FUNCTION_BLOCK FB_PrintPositionWeu EXTENDS FB_BasePrint IMPLEMENTS I_Simulation
VAR_INPUT
  IlEncoderPulse      AT%I* : UDINT;                // Encoder counter intput
  IbEncoderWcState    AT%I* : BOOL;                 // Encoder EL5101 WcState
END_VAR
VAR_OUTPUT
  bStarted                  : BOOL;                 // position started moving
  bMoving                   : BOOL;                 // position is moving
END_VAR
// ----------------------------------
// configuration
VAR
  // configuration (init)
  _fPrintResolution         : LREAL := 600;         // print(head) resolution in [dpi]
  _fSubPxResolution         : LREAL := 32;          // SubPixel resolution [SubPx], resolution factor (fI_PrintResolution*fI_SubPxResolution=>Output resolution)
  _fTaskCycleTime           : LREAL := 0.002;        // Task cycle time in [s]
END_VAR
VAR PERSISTENT
  // config values changable during runtime (recipe, visu, property)
  _fEncoderResolution       : LREAL := 1;     // Encoder resolution
END_VAR
VAR CONSTANT
  fC_MinSpeed               : LREAL := 0.05;
END_VAR
// ---------------------------------
// internal variables
VAR
  // fb inst
  //fbPositionMaster          : FB_PositionMaster;
  Fb_Ph_Master                : FB_POSITION_MASTER;
  Fb_Ref_Master               : FB_POSITION_MASTER;
  Fb_Aux_Master               : FB_POSITION_MASTER;
  
  // internal vars
  fEncoderReso              : LREAL;                // used encoder resolution
  rTrigMoving               : R_TRIG;
  // simulation
  _bSim                     : BOOL;
  rfTrig_Sim                : RF_TRIG;
    
  // test functions

END_VAR

rfTrig_Sim(CLK:=_bSim);
IF rfTrig_Sim.RT THEN SimEnter(); END_IF
IF rfTrig_Sim.FT THEN SimExit(); END_IF
IF _bSim THEN SimUpdate(); END_IF

// set internal used resolution
fEncoderReso := _fEncoderResolution;  

// calc position / speed
(*Reference Master (Used in Endless Mode with drift compensation)*)
(*---input---*)
Fb_Ref_Master.pI_ConversionErr       := ADR(PRG_SYSTEMBASE.lI_ConversionErr);
Fb_Ref_Master.bI_Reset               := bI_HardwareSync[ePr_PG_GROUP_1];  (*AutoReset*)
Fb_Ref_Master.lI_Reference           := lL_EncPulse[iL_I];
Fb_Ref_Master.fI_ResolutionInput     := fEncoderReso;
Fb_Ref_Master.fI_ResolutionOutPh     := iL_ResolutionPhPx[iL_I];
Fb_Ref_Master.fI_ResolutionOutSubPx  := iL_ResolutionSubPx[iL_I];

(*---call---*)
Fb_Ref_Master();


(*Aux Master (Used for machine speed info)*)
(*---input---*)
Fb_Aux_Master.pI_ConversionErr       := ADR(PRG_SYSTEMBASE.lI_ConversionErr);
Fb_Aux_Master.bI_Reset               := bI_HardwareSync[ePr_PG_GROUP_1];  (*AutoReset*)
Fb_Aux_Master.lI_Reference           := lIKp_EncPulse;
Fb_Aux_Master.fI_ResolutionInput     := fEncoderReso;
Fb_Aux_Master.fI_ResolutionOutPh     := iL_ResolutionPhPx[iL_I];
Fb_Aux_Master.fI_ResolutionOutSubPx  := iL_ResolutionSubPx[iL_I];

(*---call---*)
Fb_Aux_Master();


(*Printhead Master / Scaling from encoder pulses to subpixels*)
(*---input---*)
Fb_Ph_Master.pI_ConversionErr       := ADR(PRG_SYSTEMBASE.lI_ConversionErr);
Fb_Ph_Master.bI_Reset               := bI_HardwareSync[ePr_PG_GROUP_1];  (*AutoReset*)
Fb_Ph_Master.lI_Reference           := lL_EncPulse[iL_I];
Fb_Ph_Master.fI_ResolutionInput     := fL_ResolutionEncoder[iL_I] * fB_DriftControl[iL_I].fO_SpeedCorrectionFactor;
Fb_Ph_Master.fI_ResolutionOutPh     := iL_ResolutionPhPx[iL_I];
Fb_Ph_Master.fI_ResolutionOutSubPx  := iL_ResolutionSubPx[iL_I];

(*---call---*)
Fb_Ph_Master();


// postion status
bMoving := Fb_Ph_Master.fO_Master_Speed >= fC_MinSpeed; 
rTrigMoving(CLK:=bMoving);   // create started trigger output
bStarted := rTrigMoving.Q; //OR Fb_Ph_Master.bSyncReq;

PROPERTY bSimEnable : BOOL
GET
bSimEnable := _bSim;
END_GET
SET
_bSim := bSimEnable;
END_SET
END_PROPERTY

(*
  Get current "default" position.
  [SubPx] as return value and [um] as output
  :return: position in SubPx resolution
*)
METHOD getPosition : DINT
VAR_OUTPUT
  nPosition_px       : DINT;                 // Master position in [px]
  fPosition_um       : LREAL;                // Master position in [um]
END_VAR
getPosition := fbPositionMaster.lMasterPosition;
nPosition_px := fbPositionMaster.lMasterPosition / LREAL_TO_DINT(_fSubPxResolution);
fPosition_um := fbPositionMaster.fMasterPosition;
END_METHOD

(*
  Get "default" speed.
*)
METHOD getSpeed : LREAL
getSpeed := fbPositionMaster.fMasterSpeed;
END_METHOD

METHOD Init : BOOL
VAR_INPUT
  fPrintResolution    : LREAL := 600;         // print(head) resolution in [dpi]
  fSubPxResolution    : LREAL := 32;          // SubPixel resolution [SubPx], resolution factor (fI_PrintResolution*fI_SubPxResolution=>Output resolution)
  fTaskCycleTime      : LREAL;                 // Task cycle time in [s]
END_VAR
// store config
_fPrintResolution := fPrintResolution;
_fSubPxResolution := fSubPxResolution;
_fTaskCycleTime   := fTaskCycleTime;

// init fbs
// - position master
fbPositionMaster.init(
  fI_PrintResolution:=fPrintResolution, 
  fI_SubPxResolution:=fSubPxResolution, 
  fI_TaskCycleTime:=fTaskCycleTime, 
  bI_HWEncoder:=FALSE
);
END_METHOD

METHOD reset
VAR_INPUT
END_VAR
// reset positioning system
fbPositionMaster.reset();
END_METHOD

METHOD SimEnter : BOOL
_bSim := TRUE;
fbPositionMaster.bSim := TRUE;
END_METHOD

METHOD SimExit : BOOL
_bSim := FALSE;
fbPositionMaster.bSim := FALSE;
END_METHOD

METHOD SimUpdate : BOOL
//test_OldPhMaster(bEn:=bEnTestVsOld);
END_METHOD

END_FUNCTION_BLOCK

(* stored: Version 1.1.0.1, ProductVersion 3.1.4024.9
   POU FB_PrintPositionWeu: Id {726347b1-24f3-41dd-8d38-18de7bf18c3b}, SpecialFunc None
   Folder I_Simulation: Id {c1a12b52-feac-46ab-b12a-ebb95261e645}
   Property bSimEnable: Id {30fe551a-b50f-4bf8-9016-a91da26e946e}
   Get Get: Id {090ecbf3-b86f-44c9-8fdc-e451b7a045c5}
   Set Set: Id {184d9067-da40-4094-b303-24bea6510207}
   Method getPosition: Id {f3e3b96b-183e-4641-b112-e525c3bb6c11}
   Method getSpeed: Id {89c2b88d-36bc-48c9-87d7-952cfd236342}
   Method Init: Id {0edf7ce9-df28-43fb-8910-213c45b50fdb}
   Method reset: Id {2192cbfc-67ef-40f5-ae03-86c2f311383b}
   Method SimEnter: Id {18dac86d-19ba-4d47-91ad-308f9520a467}
   Method SimExit: Id {82b36d9c-34f8-4e76-b748-6f9668c98474}
   Method SimUpdate: Id {fde6f37f-ac02-4cf3-9a0e-3488a85e6ee5} *)
